///EL1259 | XFC, 8-channel digital input + 8-channel digital output with Time-Stamp
FUNCTION_BLOCK EL1259_v0_00

END_FUNCTION_BLOCK

(* stored: Version 1.1.0.1, ProductVersion 3.1.4022.6
   POU EL1259_v0_00: Id {784cd4b7-4aaf-4be9-af35-9d5415a0fb4e}, SpecialFunc None *)
